TYPE
    TcoSmartFunctionKitResults_v_4_x_x :
    STRUCT
        id : STRING;
        maxForce : REAL;
        maxPosition : REAL;
        valid : BOOL;
        createdDate : DATE;
        cycleTime : REAL;
        validationTime : INT;
        status : STRING;
        customId : STRING;
        dataRecordingDisabled : BOOL;
        samplingInterval : INT;
        _v : INT;
    END_STRUCT
END_TYPE

(* stored: Version 1.1.0.1, ProductVersion 3.1.4024.11
   DUT TcoSmartFunctionKitResults_v_4_x_x: Id {0ebb6877-3cce-41e1-861d-57af02882eb1} *)
